{attribute 'linkalways'} 
{attribute 'no_explicit_call' := 'This FB is a CLASS and must be accessed using methods or properties'}
{attribute 'enable_dynamic_creation'}
FUNCTION_BLOCK ChunkableServerResponse IMPLEMENTS I_ServerResponse
VAR
	serverResponse : I_ServerResponse;
	chunkedResponseManager : I_ChunkedResponseManager;
END_VAR

METHOD PUBLIC Accepted
VAR_INPUT
END_VAR
serverResponse.Accepted();
END_METHOD

METHOD PUBLIC Busy
VAR_INPUT
END_VAR
serverResponse.Busy();
END_METHOD

METHOD PUBLIC Error
VAR_INPUT
	ErrorCode : T_MAXSTRING;
	Message : T_MAXSTRING;
END_VAR
serverResponse.Error(ErrorCode, Message);
END_METHOD

METHOD FB_init : BOOL
VAR_INPUT
	bInitRetains : BOOL; // if TRUE, the retain variables are initialized (warm start / cold start)
	bInCopyCode : BOOL;  // if TRUE, the instance afterwards gets moved into the copy code (online change)
	ServerResponse : I_ServerResponse;
	ChunkedResponseManager : I_ChunkedResponseManager;
END_VAR
THIS^.serverResponse := ServerResponse;
This^.chunkedResponseManager := ChunkedResponseManager;
END_METHOD

PROPERTY PUBLIC Header : I_Header
GET
Header := serverResponse.Header;
END_GET
END_PROPERTY

PROPERTY PUBLIC HeadersSent : BOOL
GET
HeadersSent := serverResponse.HeadersSent;
END_GET
END_PROPERTY

METHOD PUBLIC Pending
VAR_INPUT
	ResponseId : REFERENCE TO T_MAXSTRING;
	RetryDelayInMs : UDINT;
END_VAR
serverResponse.Pending(ResponseId, RetryDelayInMs);
END_METHOD

METHOD PUBLIC Success
VAR_INPUT
END_VAR
serverResponse.Success();
END_METHOD

METHOD PUBLIC SuccessWithPayload
VAR_INPUT
	PayloadDataAddress : PVOID;
	PayloadDataSize : UDINT;
END_VAR
chunkedResponseManager.HandleSuccessWithPayload(serverResponse, PayloadDataAddress, PayloadDataSize);
END_METHOD

END_FUNCTION_BLOCK

(* stored: Version 1.1.0.1, ProductVersion 3.1.4026.13
   POU ChunkableServerResponse: Id {b8a87378-a6c1-44b3-bc88-ecbb441354ec}, SpecialFunc None
   Folder Constructor: Id {00bc04e2-5b61-4d11-87c9-cb5bcb7645f3}
   Method Accepted: Id {307f7516-cc5d-4c19-ba88-bf7819aa02e5}
   Method Busy: Id {4b537513-1564-40d9-a444-90a45308454d}
   Method Error: Id {5afbc672-088f-4657-a37c-b7486309a5f9}
   Method FB_init: Id {660d1fae-b37c-4146-aa61-1eae08e39ffd}
   Property Header: Id {235c7cc1-ede3-4dbf-bb7c-fb58221113a9}
   Get Get: Id {4a8721cf-7f0a-4d10-852a-568112ed2bdb}
   Property HeadersSent: Id {643db8fd-47fd-47d4-b4d4-78234810427d}
   Get Get: Id {d026ee17-6e55-4562-9aac-21def54df125}
   Method Pending: Id {3997d0cc-2f24-4903-a56b-9f0115921ed9}
   Method Success: Id {6890f78a-9336-404b-ba14-da4d5196941b}
   Method SuccessWithPayload: Id {b00908a6-5ec9-46cd-bdf3-9393f15ed344} *)
